PROGRAM MAIN
VAR
	bEnable : BOOL;
	
	bStart: BOOL; 
END_VAR

bEnable := bStart;

END_PROGRAM

(* stored: Version 1.1.0.1, ProductVersion 3.1.4024.12
   POU MAIN: Id {04688b04-83d1-4a1e-a4b9-dfb476a48a36}, SpecialFunc None *)
